// TIA Portal project "queueOfItems(Counters)" (V17)
// Vorlageprojekt für das Buch mit Zielsystem S7-1200

(* hardware
DEVICE "S7-1200-Station_1"  S7-1200 Station
   slot 0: "Baugruppenträger_0"  Rack  V1.0
   slot 1: "PLC_1"  CPU 1211C DC/DC/DC  6ES7 211-1AE40-0XB0  V4.1
*)

// ===== PLC "PLC_1"  CPU 1211C DC/DC/DC =====

VAR_GLOBAL   // PLC tag table "Standard-Variablentabelle"
   "itemReady" AT %I0.0 : Bool;
   "atEntry" AT %I0.1 : Bool;
   "atExit" AT %I0.2 : Bool;
   "factoryIORunning" AT %I0.3 : Bool;
   "entryConveyor" AT %Q0.0 : Bool;
   "bufferConveyor" AT %Q0.1 : Bool;
   "entryStatus" AT %M0.0 : Bool;
   "resetCounter" AT %M0.1 : Bool;
   "Tag_2" AT %M0.2 : Bool;
   "resetCounter2" AT %M0.3 : Bool;
   "Tag_3" AT %M0.7 : Bool;
   "Tag_4" AT %M0.6 : Bool;
   "loop" AT %M1.1 : Bool;
END_VAR

DATA_BLOCK "Data_block_1"   // DB3
{ S7_Optimized_Access := 'TRUE' }
VERSION : 0.1
   VAR
      counterVal : Int := 3;
   END_VAR
BEGIN
END_DATA_BLOCK

// folder: System blocks/Program resources

DATA_BLOCK "counter1"   // DB1
{ S7_Optimized_Access := 'TRUE' }
AUTHOR : Simatic
FAMILY : IEC
NAME : CNTR
VERSION : 1.0
// stored: InstanceOfName IEC_COUNTER
"IEC_COUNTER"
BEGIN
END_DATA_BLOCK

DATA_BLOCK "counter2"   // DB2
{ S7_Optimized_Access := 'TRUE' }
AUTHOR : Simatic
FAMILY : IEC
NAME : CNTR
VERSION : 1.0
// stored: InstanceOfName IEC_COUNTER
"IEC_COUNTER"
BEGIN
END_DATA_BLOCK

// folder: (top level)

FUNCTION "MHJ-PLC-Lab-Function-S71200" : Void   // FC9000, SCL
{ S7_Optimized_Access := 'TRUE' }
VERSION : 0.1
   VAR_TEMP
      rdTimeReturn : Int;
      outputTime : DTL;
      SyncVal : Byte;
      forVal : Int;
      forVal_2 : Int;
      Value : Byte;
   END_VAR
   VAR CONSTANT
      CompVal : Byte := 16#34;
      Value_01 : Byte := 16#11;
      Value_01_DW : DWord := 16#A165_D992;
      Value_02_DW : DWord := 16#58BE_4401;
   END_VAR
BEGIN

   #Value:=PEEK(area := 16#82,
        dbNumber := 0,
        byteOffset := 511);
   #Value := #Value + 1;

   POKE(area := 16#82,
        dbNumber := 0,
        byteOffset := 511,
        value := #Value);

   POKE(area:=16#81,
        dbNumber:=0,
        byteOffset:=1016,
        value:=#Value_01_DW);
   POKE(area := 16#81,
        dbNumber := 0,
        byteOffset := 1020,
        value := #Value_02_DW);

   POKE(area := 16#81,
        dbNumber := 0,
        byteOffset := 511,
        value := B#16#00);

   FOR #forVal := 0 TO 120 DO
       FOR #forVal_2:=0 TO 10 DO
           #rdTimeReturn:=RD_SYS_T(#outputTime);
           #rdTimeReturn := WR_SYS_T(#outputTime);
           #rdTimeReturn := RD_SYS_T(#outputTime);
           #rdTimeReturn := WR_SYS_T(#outputTime);
       END_FOR;
       #SyncVal:= PEEK(area := 16#81,
                      dbNumber := 0,
                      byteOffset := 511);
       IF #SyncVal = #CompVal THEN
          GOTO M_1;
       END_IF;
   END_FOR;
   RETURN;

   M_1:
   POKE(area := 16#81,
        dbNumber := 0,
        byteOffset := 511,
        value := B#16#0);
END_FUNCTION

ORGANIZATION_BLOCK "Main"   // OB1, LAD, ProgramCycle
TITLE = "Main Program Sweep (Cycle)"
{ S7_Optimized_Access := 'TRUE' }
VERSION : 0.1
   VAR_INPUT
      Initial_Call : Bool;   // Initial call of this OB
      Remanence : Bool;   // =True, if remanent data are available
   END_VAR
BEGIN

REGION Network 1: Konnektierungsbaustein für PLC-Lab
   // Im Netzwerk 1 wird der Konnektierungsbaustein für PLC-Lab aufgerufen.
   // Dieser Aufruf darf nicht entfernt werden!
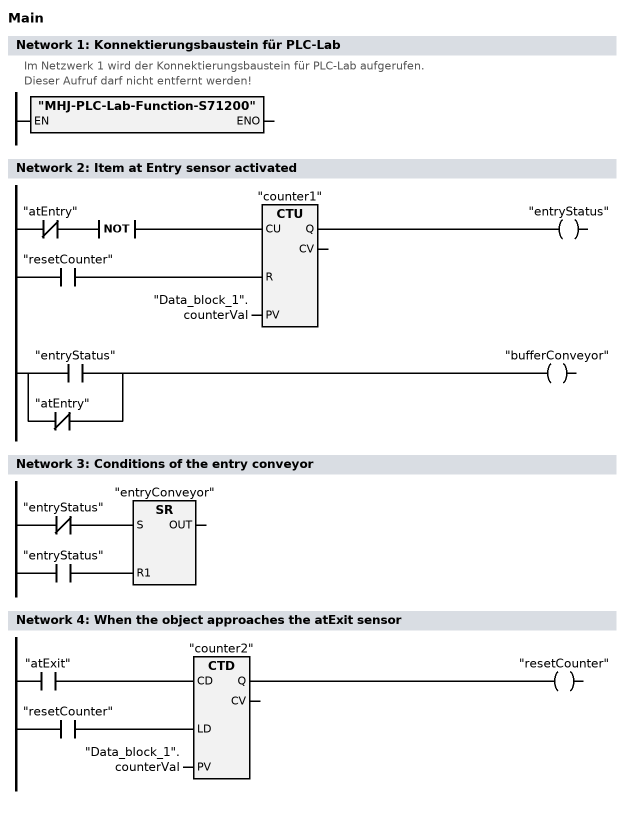
   RUNG wire#powerrail
      "MHJ-PLC-Lab-Function-S71200"()
   END_RUNG
   // the same network as SCL:
   "MHJ-PLC-Lab-Function-S71200"();
END_REGION

REGION Network 2: Item at Entry sensor activated
   "counter1".CTU(CU := NOT (NOT "atEntry"), R := "resetCounter", PV := "Data_block_1".counterVal);
   "entryStatus" := "counter1".Q;
   "bufferConveyor" := "entryStatus" OR NOT "atEntry";
END_REGION

REGION Network 3: Conditions of the entry conveyor
   RUNG wire#powerrail
      I_Contact( "entryStatus" )
      S_SR(operand := "entryConveyor", r1 := wire#w1)
   END_RUNG
   RUNG wire#powerrail
      Contact( "entryStatus" )
   END_RUNG wire#w1
   // the same network as SCL:
   IF NOT "entryStatus" THEN
       "entryConveyor" := TRUE;   // SR flip-flop
   END_IF;
   IF "entryStatus" THEN "entryConveyor" := FALSE; END_IF;
END_REGION

REGION Network 4: When the object approaches the atExit sensor
   "counter2".CTD(CD := "atExit", LD := "resetCounter", PV := "Data_block_1".counterVal);
   "resetCounter" := "counter2".Q;
END_REGION
END_ORGANIZATION_BLOCK